{attribute addProperty BoxType "EL2212-0000-0018"}
{attribute addProperty Id "DOX_Status_ChannelAT %I*ARRAY[0..1] OF DOX_Status_Channel_794B33A63240DOX_Control_ChannelAT %Q*ARRAY[0..1] OF DOX_Control_Channel_0C4BF1873240WcStateAT %I*WcState_98A4DF7520.250InfoDataAT %I*InfoData_BC63D37F80100"}
{attribute addProperty CRC "3262838998"}
{attribute addProperty SizeInBites "146"}
{attribute addProperty SizeInBytes "18.25"}
TYPE EL2212_74FAECA9 :
STRUCT
	{attribute addProperty Name "DOX_Status_Channel"}
	DOX_Status_Channel : ARRAY[0..1] OF DOX_Status_Channel_794B33A6;
	{attribute addProperty Name "DOX_Control_Channel"}
	DOX_Control_Channel : ARRAY[0..1] OF DOX_Control_Channel_0C4BF187;
	{attribute addProperty Name "WcState"}
	WcState : WcState_98A4DF75;
	{attribute addProperty Name "InfoData"}
	InfoData : InfoData_BC63D37F;
END_STRUCT
END_TYPE

(* stored: Version 1.2.0.0, ProductVersion 3.1.4024.9
   DUT EL2212_74FAECA9: Id {b97b4108-d10f-4734-9e36-dc398d95be81} *)
